// TIA Portal V18 export
// export: Created 2026-04-18T00:00:00Z, ExportSetting WithDefaults
FUNCTION "FC_Init_Default_Recipe_PLC2" : Void   // FC51, LAD
{ S7_Optimized_Access := 'TRUE' }
VERSION : 0.1
// stored: AutoNumber true, IsIECCheckEnabled false
BEGIN

REGION Network 1: Kích hoạt nạp recipe mặc định lần đầu scan PLC2
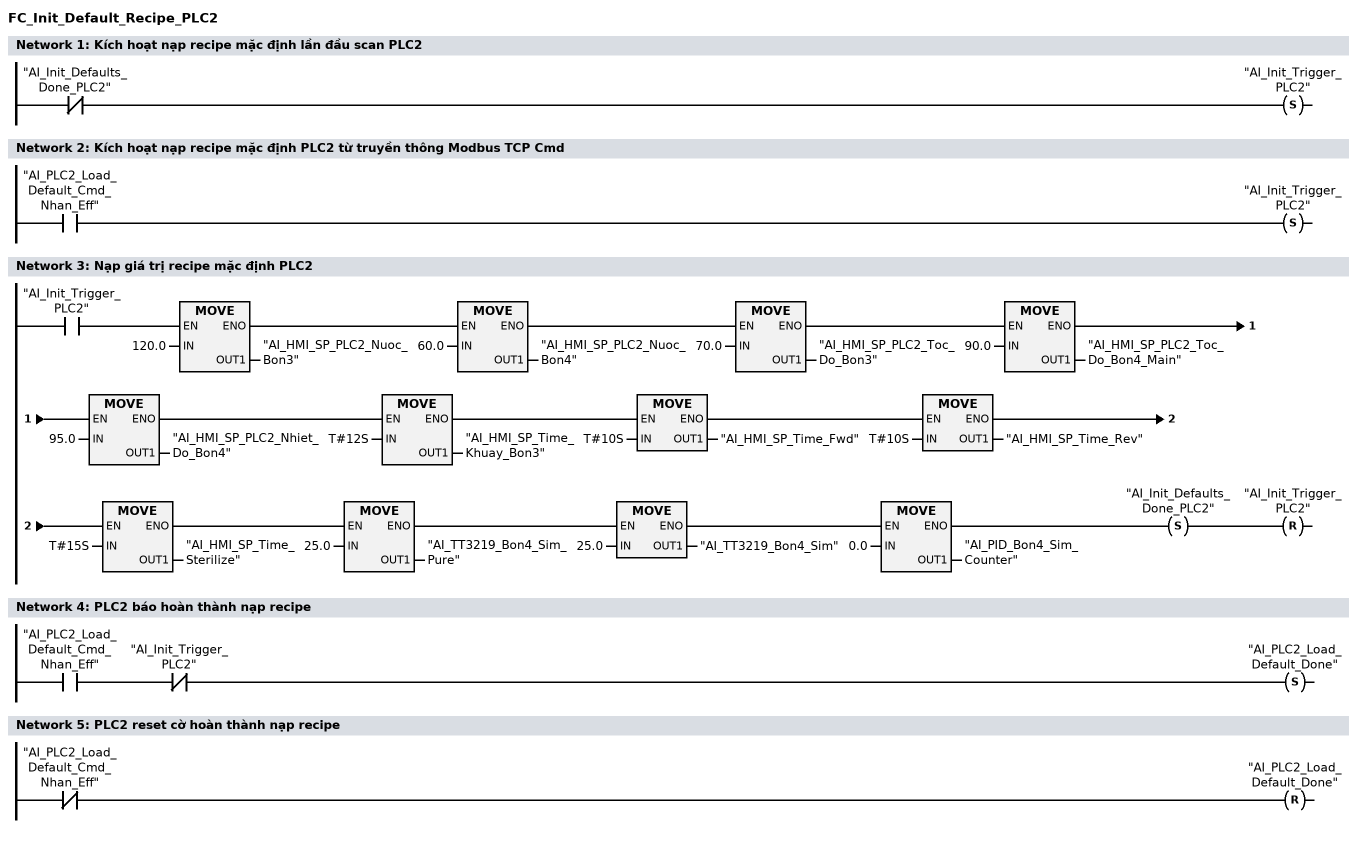
   RUNG wire#powerrail
      I_Contact( "AI_Init_Defaults_Done_PLC2" )
      S_Coil( "AI_Init_Trigger_PLC2" )
   END_RUNG
   // the same network as SCL:
   IF NOT "AI_Init_Defaults_Done_PLC2" THEN "AI_Init_Trigger_PLC2" := TRUE; END_IF;
END_REGION

REGION Network 2: Kích hoạt nạp recipe mặc định PLC2 từ truyền thông Modbus TCP Cmd
   RUNG wire#powerrail
      Contact( "AI_PLC2_Load_Default_Cmd_Nhan_Eff" )
      S_Coil( "AI_Init_Trigger_PLC2" )
   END_RUNG
   // the same network as SCL:
   IF "AI_PLC2_Load_Default_Cmd_Nhan_Eff" THEN "AI_Init_Trigger_PLC2" := TRUE; END_IF;
END_REGION

REGION Network 3: Nạp giá trị recipe mặc định PLC2
   RUNG wire#powerrail
      Contact( "AI_Init_Trigger_PLC2" )
      { S7_GenerateENO := "TRUE" } Move(in := 120.0, out1 => "AI_HMI_SP_PLC2_Nuoc_Bon3")
      { S7_GenerateENO := "TRUE" } Move(in := 60.0, out1 => "AI_HMI_SP_PLC2_Nuoc_Bon4")
      { S7_GenerateENO := "TRUE" } Move(in := 70.0, out1 => "AI_HMI_SP_PLC2_Toc_Do_Bon3")
      { S7_GenerateENO := "TRUE" } Move(in := 90.0, out1 => "AI_HMI_SP_PLC2_Toc_Do_Bon4_Main")
      { S7_GenerateENO := "TRUE" } Move(in := 95.0, out1 => "AI_HMI_SP_PLC2_Nhiet_Do_Bon4")
      { S7_GenerateENO := "TRUE" } Move(in := T#12S, out1 => "AI_HMI_SP_Time_Khuay_Bon3")
      { S7_GenerateENO := "TRUE" } Move(in := T#10S, out1 => "AI_HMI_SP_Time_Fwd")
      { S7_GenerateENO := "TRUE" } Move(in := T#10S, out1 => "AI_HMI_SP_Time_Rev")
      { S7_GenerateENO := "TRUE" } Move(in := T#15S, out1 => "AI_HMI_SP_Time_Sterilize")
      { S7_GenerateENO := "TRUE" } Move(in := 25.0, out1 => "AI_TT3219_Bon4_Sim_Pure")
      { S7_GenerateENO := "TRUE" } Move(in := 25.0, out1 => "AI_TT3219_Bon4_Sim")
      { S7_GenerateENO := "TRUE" } Move(in := 0.0, out1 => "AI_PID_Bon4_Sim_Counter")
      S_Coil( "AI_Init_Defaults_Done_PLC2" )
      R_Coil( "AI_Init_Trigger_PLC2" )
   END_RUNG
   // the same network as SCL:
   // ENO of a box is taken as its EN; it also drops when the box reports an error
   IF "AI_Init_Trigger_PLC2" THEN
       "AI_HMI_SP_PLC2_Nuoc_Bon3" := 120.0;
       "AI_HMI_SP_PLC2_Nuoc_Bon4" := 60.0;
       "AI_HMI_SP_PLC2_Toc_Do_Bon3" := 70.0;
       "AI_HMI_SP_PLC2_Toc_Do_Bon4_Main" := 90.0;
       "AI_HMI_SP_PLC2_Nhiet_Do_Bon4" := 95.0;
       "AI_HMI_SP_Time_Khuay_Bon3" := T#12S;
       "AI_HMI_SP_Time_Fwd" := T#10S;
       "AI_HMI_SP_Time_Rev" := T#10S;
       "AI_HMI_SP_Time_Sterilize" := T#15S;
       "AI_TT3219_Bon4_Sim_Pure" := 25.0;
       "AI_TT3219_Bon4_Sim" := 25.0;
       "AI_PID_Bon4_Sim_Counter" := 0.0;
       "AI_Init_Defaults_Done_PLC2" := TRUE;
       "AI_Init_Trigger_PLC2" := FALSE;
   END_IF;
END_REGION

REGION Network 4: PLC2 báo hoàn thành nạp recipe
   RUNG wire#powerrail
      Contact( "AI_PLC2_Load_Default_Cmd_Nhan_Eff" )
      I_Contact( "AI_Init_Trigger_PLC2" )
      S_Coil( "AI_PLC2_Load_Default_Done" )
   END_RUNG
   // the same network as SCL:
   IF "AI_PLC2_Load_Default_Cmd_Nhan_Eff" AND NOT "AI_Init_Trigger_PLC2" THEN
       "AI_PLC2_Load_Default_Done" := TRUE;
   END_IF;
END_REGION

REGION Network 5: PLC2 reset cờ hoàn thành nạp recipe
   RUNG wire#powerrail
      I_Contact( "AI_PLC2_Load_Default_Cmd_Nhan_Eff" )
      R_Coil( "AI_PLC2_Load_Default_Done" )
   END_RUNG
   // the same network as SCL:
   IF NOT "AI_PLC2_Load_Default_Cmd_Nhan_Eff" THEN "AI_PLC2_Load_Default_Done" := FALSE; END_IF;
END_REGION
END_FUNCTION
